    ENDPROC
    PROC Reflejado()
        MoveL Target_x_2,v100,z1,Marcador\WObj:=Pastel_2;
        MoveL Aproximacion_2,v100,z1,Marcador\WObj:=Pastel_2;
        MoveL HOME_2,v100,z1,Marcador\WObj:=Pastel_2;
        MoveL orientacioin_posible_2,v100,z1,Marcador\WObj:=Pastel_2;
        MoveL Target_10_2,v100,z1,Marcador\WObj:=Pastel_2;
        MoveL Target_20_2,v100,z1,Marcador\WObj:=Pastel_2;
        MoveL Target_30_2,v100,z1,Marcador\WObj:=Pastel_2;
        MoveL Target_40_2,v100,z1,Marcador\WObj:=Pastel_2;
        MoveL Target_50_2,v100,z1,Marcador\WObj:=Pastel_2;
        MoveL Target_60_2,v100,z1,Marcador\WObj:=Pastel_2;
        MoveL Target_70_2,v100,z1,Marcador\WObj:=Pastel_2;
        MoveL Target_80_2,v100,z1,Marcador\WObj:=Pastel_2;
        MoveL Target_90_2,v100,z1,Marcador\WObj:=Pastel_2;
        MoveL Target_100_2,v100,z1,Marcador\WObj:=Pastel_2;
        MoveL Target_110_2,v100,z1,Marcador\WObj:=Pastel_2;
        MoveL Target_120_2,v100,z1,Marcador\WObj:=Pastel_2;
        MoveL Target_130_2,v100,z1,Marcador\WObj:=Pastel_2;
        MoveL Target_140_2,v100,z1,Marcador\WObj:=Pastel_2;
        MoveL Target_150_2,v100,z1,Marcador\WObj:=Pastel_2;
        MoveL Target_160_2,v100,z1,Marcador\WObj:=Pastel_2;
        MoveL Target_170_2,v100,z1,Marcador\WObj:=Pastel_2;
        MoveL Target_180_2,v100,z1,Marcador\WObj:=Pastel_2;
        MoveL Target_190_2,v100,z1,Marcador\WObj:=Pastel_2;
        MoveL Target_200_2,v100,z1,Marcador\WObj:=Pastel_2;
        MoveL Target_210_2,v100,z1,Marcador\WObj:=Pastel_2;
        MoveL Target_220_2,v100,z1,Marcador\WObj:=Pastel_2;
        MoveL Target_230_2,v100,z1,Marcador\WObj:=Pastel_2;
        MoveL Target_240_2,v100,z1,Marcador\WObj:=Pastel_2;
        MoveL Target_250_2,v100,z1,Marcador\WObj:=Pastel_2;
        MoveL Target_260_2,v100,z1,Marcador\WObj:=Pastel_2;
        MoveL Target_270_2,v100,z1,Marcador\WObj:=Pastel_2;
        MoveL Target_280_2,v100,z1,Marcador\WObj:=Pastel_2;
        MoveL Target_290_2,v100,z1,Marcador\WObj:=Pastel_2;
        MoveL Target_300_2,v100,z1,Marcador\WObj:=Pastel_2;
        MoveL Target_310_2,v100,z1,Marcador\WObj:=Pastel_2;
        MoveL Target_320_2,v100,z1,Marcador\WObj:=Pastel_2;
        MoveL Target_330_2,v100,z1,Marcador\WObj:=Pastel_2;
        MoveL Target_340_2,v100,z1,Marcador\WObj:=Pastel_2;
        MoveL Target_350_2,v100,z1,Marcador\WObj:=Pastel_2;
        MoveL Target_360_2,v100,z1,Marcador\WObj:=Pastel_2;
        MoveL Target_370_2,v100,z1,Marcador\WObj:=Pastel_2;
        MoveL Target_380_2,v100,z1,Marcador\WObj:=Pastel_2;
        MoveL Target_390_2,v100,z1,Marcador\WObj:=Pastel_2;
        MoveL Target_400_2,v100,z1,Marcador\WObj:=Pastel_2;
        MoveL Target_410_2,v100,z1,Marcador\WObj:=Pastel_2;
        MoveL Target_420_2,v100,z1,Marcador\WObj:=Pastel_2;
        MoveL Target_430_2,v100,z1,Marcador\WObj:=Pastel_2;
        MoveL Target_440_2,v100,z1,Marcador\WObj:=Pastel_2;
        MoveL Target_450_2,v100,z1,Marcador\WObj:=Pastel_2;
        MoveL Target_460_2,v100,z1,Marcador\WObj:=Pastel_2;
        MoveL Target_470_2,v100,z1,Marcador\WObj:=Pastel_2;
        MoveL Target_480_2,v100,z1,Marcador\WObj:=Pastel_2;
        MoveL Target_490_2,v100,z1,Marcador\WObj:=Pastel_2;
        MoveL Target_500_2,v100,z1,Marcador\WObj:=Pastel_2;
        MoveL Target_510_2,v100,z1,Marcador\WObj:=Pastel_2;
        MoveL Target_520_2,v100,z1,Marcador\WObj:=Pastel_2;
        MoveL Target_530_2,v100,z1,Marcador\WObj:=Pastel_2;
        MoveL Target_540_2,v100,z1,Marcador\WObj:=Pastel_2;
        MoveL Target_550_2,v100,z1,Marcador\WObj:=Pastel_2;
        MoveL Target_560_2,v100,z1,Marcador\WObj:=Pastel_2;
        MoveL Target_570_2,v100,z1,Marcador\WObj:=Pastel_2;
        MoveL Target_580_2,v100,z1,Marcador\WObj:=Pastel_2;
        MoveL Target_590_2,v100,z1,Marcador\WObj:=Pastel_2;
        MoveL Target_600_2,v100,z1,Marcador\WObj:=Pastel_2;
        MoveL Target_610_2,v100,z1,Marcador\WObj:=Pastel_2;
        MoveL Target_620_2,v100,z1,Marcador\WObj:=Pastel_2;
        MoveL Target_630_2,v100,z1,Marcador\WObj:=Pastel_2;
        MoveL Target_640_2,v100,z1,Marcador\WObj:=Pastel_2;
        MoveL Target_650_2,v100,z1,Marcador\WObj:=Pastel_2;
        MoveL Target_660_2,v100,z1,Marcador\WObj:=Pastel_2;
        MoveL Target_670_2,v100,z1,Marcador\WObj:=Pastel_2;
        MoveL Target_680_2,v100,z1,Marcador\WObj:=Pastel_2;
        MoveL Target_690_2,v100,z1,Marcador\WObj:=Pastel_2;
        MoveL Target_700_2,v100,z1,Marcador\WObj:=Pastel_2;
        MoveL Target_710_2,v100,z1,Marcador\WObj:=Pastel_2;
        MoveL Target_720_2,v100,z1,Marcador\WObj:=Pastel_2;
        MoveL Target_730_2,v100,z1,Marcador\WObj:=Pastel_2;
        MoveL Target_740_2,v100,z1,Marcador\WObj:=Pastel_2;
        MoveL Target_750_2,v100,z1,Marcador\WObj:=Pastel_2;
        MoveL Target_760_2,v100,z1,Marcador\WObj:=Pastel_2;
        MoveL Target_770_2,v100,z1,Marcador\WObj:=Pastel_2;
        MoveL Target_780_2,v100,z1,Marcador\WObj:=Pastel_2;
        MoveL Target_790_2,v100,z1,Marcador\WObj:=Pastel_2;
        MoveL Target_800_2,v100,z1,Marcador\WObj:=Pastel_2;
        MoveL Target_810_2,v100,z1,Marcador\WObj:=Pastel_2;
        MoveL Target_820_2,v100,z1,Marcador\WObj:=Pastel_2;
        MoveL Target_830_2,v100,z1,Marcador\WObj:=Pastel_2;
        MoveL Target_840_2,v100,z1,Marcador\WObj:=Pastel_2;
        MoveL Target_850_2,v100,z1,Marcador\WObj:=Pastel_2;
        MoveL Target_860_2,v100,z1,Marcador\WObj:=Pastel_2;
        MoveL Target_870_2,v100,z1,Marcador\WObj:=Pastel_2;
        MoveL Target_880_2,v100,z1,Marcador\WObj:=Pastel_2;
        MoveL Target_890_2,v100,z1,Marcador\WObj:=Pastel_2;
        MoveL Target_900_2,v100,z1,Marcador\WObj:=Pastel_2;
        MoveL Target_910_2,v100,z1,Marcador\WObj:=Pastel_2;
        MoveL Target_920_2,v100,z1,Marcador\WObj:=Pastel_2;
        MoveL Target_930_2,v100,z1,Marcador\WObj:=Pastel_2;
        MoveL Target_940_2,v100,z1,Marcador\WObj:=Pastel_2;
        MoveL Target_950_2,v100,z1,Marcador\WObj:=Pastel_2;
        MoveL Target_960_2,v100,z1,Marcador\WObj:=Pastel_2;
        MoveL Target_970_2,v100,z1,Marcador\WObj:=Pastel_2;
        MoveL Target_980_2,v100,z1,Marcador\WObj:=Pastel_2;
        MoveL Target_990_2,v100,z1,Marcador\WObj:=Pastel_2;
        MoveL Target_1000_2,v100,z1,Marcador\WObj:=Pastel_2;
        MoveL Target_1010_2,v100,z1,Marcador\WObj:=Pastel_2;
        MoveL Target_1020_2,v100,z1,Marcador\WObj:=Pastel_2;
        MoveL Target_1030_2,v100,z1,Marcador\WObj:=Pastel_2;
        MoveL Target_1040_2,v100,z1,Marcador\WObj:=Pastel_2;
        MoveL Target_1050_2,v100,z1,Marcador\WObj:=Pastel_2;
        MoveL Target_1060_2,v100,z1,Marcador\WObj:=Pastel_2;
        MoveL Target_1070_2,v100,z1,Marcador\WObj:=Pastel_2;
        MoveL Target_1080_2,v100,z1,Marcador\WObj:=Pastel_2;
        MoveL Target_1090_2,v100,z1,Marcador\WObj:=Pastel_2;
        MoveL Target_1100_2,v100,z1,Marcador\WObj:=Pastel_2;
        MoveL Target_1110_2,v100,z1,Marcador\WObj:=Pastel_2;
        MoveL Target_1120_2,v100,z1,Marcador\WObj:=Pastel_2;
        MoveL Target_1130_2,v100,z1,Marcador\WObj:=Pastel_2;
        MoveL Target_1140_2,v100,z1,Marcador\WObj:=Pastel_2;
        MoveL Target_1150_2,v100,z1,Marcador\WObj:=Pastel_2;
        MoveL Target_1160_2,v100,z1,Marcador\WObj:=Pastel_2;
        MoveL Target_1170_2,v100,z1,Marcador\WObj:=Pastel_2;
        MoveL Target_1180_2,v100,z1,Marcador\WObj:=Pastel_2;
        MoveL Target_1190_2,v100,z1,Marcador\WObj:=Pastel_2;
        MoveL Target_1200_2,v100,z1,Marcador\WObj:=Pastel_2;
        MoveL Target_1210_2,v100,z1,Marcador\WObj:=Pastel_2;
        MoveL Target_1220_2,v100,z1,Marcador\WObj:=Pastel_2;
        MoveL Target_1230_2,v100,z1,Marcador\WObj:=Pastel_2;
        MoveL Target_1240_2,v100,z1,Marcador\WObj:=Pastel_2;
        MoveL Target_1250_2,v100,z1,Marcador\WObj:=Pastel_2;
        MoveL Target_1260_2,v100,z1,Marcador\WObj:=Pastel_2;
        MoveL Target_1270_2,v100,z1,Marcador\WObj:=Pastel_2;
        MoveL Target_1280_2,v100,z1,Marcador\WObj:=Pastel_2;
        MoveL Target_1290_2,v100,z1,Marcador\WObj:=Pastel_2;
        MoveL Target_1300_2,v100,z1,Marcador\WObj:=Pastel_2;
        MoveL Target_1310_2,v100,z1,Marcador\WObj:=Pastel_2;
        MoveL Target_1320_2,v100,z1,Marcador\WObj:=Pastel_2;
        MoveL Target_1330_2,v100,z1,Marcador\WObj:=Pastel_2;
        MoveL Target_1340_2,v100,z1,Marcador\WObj:=Pastel_2;
        MoveL Target_1350_2,v100,z1,Marcador\WObj:=Pastel_2;
        MoveL Target_1360_2,v100,z1,Marcador\WObj:=Pastel_2;
        MoveL Target_1370_2,v100,z1,Marcador\WObj:=Pastel_2;
        MoveL Target_1380_2,v100,z1,Marcador\WObj:=Pastel_2;
        MoveL Target_1390_2,v100,z1,Marcador\WObj:=Pastel_2;
        MoveL Target_1400_2,v100,z1,Marcador\WObj:=Pastel_2;
        MoveL Target_1410_2,v100,z1,Marcador\WObj:=Pastel_2;
        MoveL Target_1420_2,v100,z1,Marcador\WObj:=Pastel_2;
        MoveL Target_1430_2,v100,z1,Marcador\WObj:=Pastel_2;
        MoveL Target_1440_2,v100,z1,Marcador\WObj:=Pastel_2;
        MoveL Target_1450_2,v100,z1,Marcador\WObj:=Pastel_2;
        MoveL Target_1460_2,v100,z1,Marcador\WObj:=Pastel_2;
        MoveL Target_1470_2,v100,z1,Marcador\WObj:=Pastel_2;
        MoveL Target_1480_2,v100,z1,Marcador\WObj:=Pastel_2;
        MoveL Target_1490_2,v100,z1,Marcador\WObj:=Pastel_2;
        MoveL Target_1500_2,v100,z1,Marcador\WObj:=Pastel_2;
        MoveL Target_1510_2,v100,z1,Marcador\WObj:=Pastel_2;
        MoveL Target_1520_2,v100,z1,Marcador\WObj:=Pastel_2;
        MoveL Target_1530_2,v100,z1,Marcador\WObj:=Pastel_2;
        MoveL Target_1540_2,v100,z1,Marcador\WObj:=Pastel_2;
        MoveL Target_1550_2,v100,z1,Marcador\WObj:=Pastel_2;
        MoveL Target_1560_2,v100,z1,Marcador\WObj:=Pastel_2;
        MoveL Target_1570_2,v100,z1,Marcador\WObj:=Pastel_2;
        MoveL Target_1580_2,v100,z1,Marcador\WObj:=Pastel_2;
        MoveL Target_1590_2,v100,z1,Marcador\WObj:=Pastel_2;
        MoveL Target_1600_2,v100,z1,Marcador\WObj:=Pastel_2;
        MoveL Target_1610_2,v100,z1,Marcador\WObj:=Pastel_2;
        MoveL Target_1620_2,v100,z1,Marcador\WObj:=Pastel_2;
        MoveL Target_1630_2,v100,z1,Marcador\WObj:=Pastel_2;
        MoveL Target_1640_2,v100,z1,Marcador\WObj:=Pastel_2;
        MoveL Target_1650_2,v100,z1,Marcador\WObj:=Pastel_2;
        MoveL Target_1660_2,v100,z1,Marcador\WObj:=Pastel_2;
        MoveL Target_1670_2,v100,z1,Marcador\WObj:=Pastel_2;
        MoveL Target_1680_2,v100,z1,Marcador\WObj:=Pastel_2;
        MoveL Target_1690_2,v100,z1,Marcador\WObj:=Pastel_2;
        MoveL Target_1700_2,v100,z1,Marcador\WObj:=Pastel_2;
        MoveL Target_1710_2,v100,z1,Marcador\WObj:=Pastel_2;
        MoveL Target_1720_2,v100,z1,Marcador\WObj:=Pastel_2;
        MoveL Target_1730_2,v100,z1,Marcador\WObj:=Pastel_2;
        MoveL Target_1740_2,v100,z1,Marcador\WObj:=Pastel_2;
        MoveL Target_1750_2,v100,z1,Marcador\WObj:=Pastel_2;
        MoveL Target_1760_2,v100,z1,Marcador\WObj:=Pastel_2;
        MoveL Target_1770_2,v100,z1,Marcador\WObj:=Pastel_2;
        MoveL Target_1780_2,v100,z1,Marcador\WObj:=Pastel_2;
        MoveL Target_1790_2,v100,z1,Marcador\WObj:=Pastel_2;
        MoveL Target_1800_2,v100,z1,Marcador\WObj:=Pastel_2;
        MoveL Target_1810_2,v100,z1,Marcador\WObj:=Pastel_2;
        MoveL Target_1820_2,v100,z1,Marcador\WObj:=Pastel_2;
        MoveL Target_1830_2,v100,z1,Marcador\WObj:=Pastel_2;
        MoveL Target_1840_2,v100,z1,Marcador\WObj:=Pastel_2;
        MoveL Target_1850_2,v100,z1,Marcador\WObj:=Pastel_2;
        MoveL Target_1860_2,v100,z1,Marcador\WObj:=Pastel_2;
        MoveL Target_1870_2,v100,z1,Marcador\WObj:=Pastel_2;
        MoveL Target_1880_2,v100,z1,Marcador\WObj:=Pastel_2;
        MoveL Target_1890_2,v100,z1,Marcador\WObj:=Pastel_2;
        MoveL Target_1900_2,v100,z1,Marcador\WObj:=Pastel_2;
        MoveL Target_1910_2,v100,z1,Marcador\WObj:=Pastel_2;
        MoveL Target_1920_2,v100,z1,Marcador\WObj:=Pastel_2;
        MoveL Target_1930_2,v100,z1,Marcador\WObj:=Pastel_2;
        MoveL Target_1940_2,v100,z1,Marcador\WObj:=Pastel_2;
        MoveL Target_1950_2,v100,z1,Marcador\WObj:=Pastel_2;
        MoveL Target_1960_2,v100,z1,Marcador\WObj:=Pastel_2;
        MoveL Target_1970_2,v100,z1,Marcador\WObj:=Pastel_2;
        MoveL Target_1980_2,v100,z1,Marcador\WObj:=Pastel_2;
        MoveL Target_1990_2,v100,z1,Marcador\WObj:=Pastel_2;
        MoveL Target_2000_2,v100,z1,Marcador\WObj:=Pastel_2;
        MoveL Target_2010_2,v100,z1,Marcador\WObj:=Pastel_2;
        MoveL Target_2020_2,v100,z1,Marcador\WObj:=Pastel_2;
        MoveL Target_2030_2,v100,z1,Marcador\WObj:=Pastel_2;
        MoveL Target_2040_2,v100,z1,Marcador\WObj:=Pastel_2;
        MoveL Target_2050_2,v100,z1,Marcador\WObj:=Pastel_2;
        MoveL Target_2060_2,v100,z1,Marcador\WObj:=Pastel_2;
        MoveL Target_2070_2,v100,z1,Marcador\WObj:=Pastel_2;
        MoveL Target_2080_2,v100,z1,Marcador\WObj:=Pastel_2;
        MoveL Target_2090_2,v100,z1,Marcador\WObj:=Pastel_2;
        MoveL Target_2100_2,v100,z1,Marcador\WObj:=Pastel_2;
        MoveL Target_2110_2,v100,z1,Marcador\WObj:=Pastel_2;
        MoveL Target_2120_2,v100,z1,Marcador\WObj:=Pastel_2;
        MoveL Target_2130_2,v100,z1,Marcador\WObj:=Pastel_2;
        MoveL Target_2140_2,v100,z1,Marcador\WObj:=Pastel_2;
        MoveL Target_2150_2,v100,z1,Marcador\WObj:=Pastel_2;
        MoveL Target_2160_2,v100,z1,Marcador\WObj:=Pastel_2;
        MoveL Target_2170_2,v100,z1,Marcador\WObj:=Pastel_2;
        MoveL Target_2180_2,v100,z1,Marcador\WObj:=Pastel_2;
        MoveL Target_2190_2,v100,z1,Marcador\WObj:=Pastel_2;
        MoveL Target_2200_2,v100,z1,Marcador\WObj:=Pastel_2;
        MoveL Target_2210_2,v100,z1,Marcador\WObj:=Pastel_2;
        MoveL Target_2220_2,v100,z1,Marcador\WObj:=Pastel_2;
        MoveL Target_2230_2,v100,z1,Marcador\WObj:=Pastel_2;
        MoveL Target_2240_2,v100,z1,Marcador\WObj:=Pastel_2;
        MoveL Target_2250_2,v100,z1,Marcador\WObj:=Pastel_2;
        MoveL Target_2260_2,v100,z1,Marcador\WObj:=Pastel_2;
        MoveL Target_2270_2,v100,z1,Marcador\WObj:=Pastel_2;
        MoveL Target_2280_2,v100,z1,Marcador\WObj:=Pastel_2;
        MoveL Target_2290_2,v100,z1,Marcador\WObj:=Pastel_2;
        MoveL Target_2300_2,v100,z1,Marcador\WObj:=Pastel_2;
        MoveL Target_2310_2,v100,z1,Marcador\WObj:=Pastel_2;
        MoveL Target_2320_2,v100,z1,Marcador\WObj:=Pastel_2;
        MoveL Target_2330_2,v100,z1,Marcador\WObj:=Pastel_2;
        MoveL Target_2340_2,v100,z1,Marcador\WObj:=Pastel_2;
        MoveL Target_2350_2,v100,z1,Marcador\WObj:=Pastel_2;
        MoveL Target_2360_2,v100,z1,Marcador\WObj:=Pastel_2;
        MoveL Target_2370_2,v100,z1,Marcador\WObj:=Pastel_2;
        MoveL Target_2380_2,v100,z1,Marcador\WObj:=Pastel_2;
        MoveL Target_2390_2,v100,z1,Marcador\WObj:=Pastel_2;
        MoveL Target_2400_2,v100,z1,Marcador\WObj:=Pastel_2;
        MoveL Target_2410_2,v100,z1,Marcador\WObj:=Pastel_2;
        MoveL Target_2420_2,v100,z1,Marcador\WObj:=Pastel_2;
        MoveL Target_2430_2,v100,z1,Marcador\WObj:=Pastel_2;
        MoveL Target_2440_2,v100,z1,Marcador\WObj:=Pastel_2;
        MoveL Target_2450_2,v100,z1,Marcador\WObj:=Pastel_2;
        MoveL Target_2460_2,v100,z1,Marcador\WObj:=Pastel_2;
        MoveL Target_2470_2,v100,z1,Marcador\WObj:=Pastel_2;
        MoveL Target_2480_2,v100,z1,Marcador\WObj:=Pastel_2;
        MoveL Target_2490_2,v100,z1,Marcador\WObj:=Pastel_2;
        MoveL Target_2500_2,v100,z1,Marcador\WObj:=Pastel_2;
        MoveL Target_2510_2,v100,z1,Marcador\WObj:=Pastel_2;
        MoveL Target_2520_2,v100,z1,Marcador\WObj:=Pastel_2;
        MoveL Target_2530_2,v100,z1,Marcador\WObj:=Pastel_2;
        MoveL Target_2540_2,v100,z1,Marcador\WObj:=Pastel_2;
        MoveL Target_2550_2,v100,z1,Marcador\WObj:=Pastel_2;
        MoveL Target_2560_2,v100,z1,Marcador\WObj:=Pastel_2;
        MoveL Target_2570_2,v100,z1,Marcador\WObj:=Pastel_2;
        MoveL Target_2580_2,v100,z1,Marcador\WObj:=Pastel_2;
        MoveL Target_2590_2,v100,z1,Marcador\WObj:=Pastel_2;
        MoveL Target_2600_2,v100,z1,Marcador\WObj:=Pastel_2;
        MoveL Target_2610_2,v100,z1,Marcador\WObj:=Pastel_2;
        MoveL Target_2620_2,v100,z1,Marcador\WObj:=Pastel_2;
        MoveL Target_2630_2,v100,z1,Marcador\WObj:=Pastel_2;
        MoveL Target_2640_2,v100,z1,Marcador\WObj:=Pastel_2;
        MoveL Target_2650_2,v100,z1,Marcador\WObj:=Pastel_2;
        MoveL Target_2660_2,v100,z1,Marcador\WObj:=Pastel_2;
        MoveL Target_2670_2,v100,z1,Marcador\WObj:=Pastel_2;
        MoveL Target_2680_2,v100,z1,Marcador\WObj:=Pastel_2;
        MoveL Target_2690_2,v100,z1,Marcador\WObj:=Pastel_2;
        MoveL Target_2700_2,v100,z1,Marcador\WObj:=Pastel_2;
        MoveL Target_2710_2,v100,z1,Marcador\WObj:=Pastel_2;
        MoveL Target_2720_2,v100,z1,Marcador\WObj:=Pastel_2;
        MoveL Target_2730_2,v100,z1,Marcador\WObj:=Pastel_2;
        MoveL Target_2740_2,v100,z1,Marcador\WObj:=Pastel_2;
        MoveL Target_2750_2,v100,z1,Marcador\WObj:=Pastel_2;
        MoveL Target_2760_2,v100,z1,Marcador\WObj:=Pastel_2;
        MoveL Target_2770_2,v100,z1,Marcador\WObj:=Pastel_2;
        MoveL Target_2780_2,v100,z1,Marcador\WObj:=Pastel_2;
        MoveL Target_2790_2,v100,z1,Marcador\WObj:=Pastel_2;
        MoveL Target_2800_2,v100,z1,Marcador\WObj:=Pastel_2;
        MoveL Target_2810_2,v100,z1,Marcador\WObj:=Pastel_2;
        MoveL Target_2820_2,v100,z1,Marcador\WObj:=Pastel_2;
        MoveL Target_2830_2,v100,z1,Marcador\WObj:=Pastel_2;
        MoveL Target_2840_2,v100,z1,Marcador\WObj:=Pastel_2;
        MoveL Target_2850_2,v100,z1,Marcador\WObj:=Pastel_2;
        MoveL Target_2860_2,v100,z1,Marcador\WObj:=Pastel_2;
        MoveL Target_2870_2,v100,z1,Marcador\WObj:=Pastel_2;
        MoveL Target_2880_2,v100,z1,Marcador\WObj:=Pastel_2;
        MoveL Target_2890_2,v100,z1,Marcador\WObj:=Pastel_2;
        MoveL Target_2900_2,v100,z1,Marcador\WObj:=Pastel_2;
        MoveL Target_2910_2,v100,z1,Marcador\WObj:=Pastel_2;
        MoveL Target_2920_2,v100,z1,Marcador\WObj:=Pastel_2;
        MoveL Target_2930_2,v100,z1,Marcador\WObj:=Pastel_2;
        MoveL Target_2940_2,v100,z1,Marcador\WObj:=Pastel_2;
        MoveL Target_2950_2,v100,z1,Marcador\WObj:=Pastel_2;
        MoveL Target_2960_2,v100,z1,Marcador\WObj:=Pastel_2;
        MoveL Target_2970_2,v100,z1,Marcador\WObj:=Pastel_2;
        MoveL Target_2980_2,v100,z1,Marcador\WObj:=Pastel_2;
        MoveL Target_2990_2,v100,z1,Marcador\WObj:=Pastel_2;
        MoveL Target_3000_2,v100,z1,Marcador\WObj:=Pastel_2;
        MoveL Target_3010_2,v100,z1,Marcador\WObj:=Pastel_2;
        MoveL Target_3020_2,v100,z1,Marcador\WObj:=Pastel_2;
        MoveL Target_3030_2,v100,z1,Marcador\WObj:=Pastel_2;
        MoveL Target_3040_2,v100,z1,Marcador\WObj:=Pastel_2;
        MoveL Target_3050_2,v100,z1,Marcador\WObj:=Pastel_2;
        MoveL Target_3060_2,v100,z1,Marcador\WObj:=Pastel_2;
        MoveL Target_3070_2,v100,z1,Marcador\WObj:=Pastel_2;
        MoveL Target_3080_2,v100,z1,Marcador\WObj:=Pastel_2;
        MoveL Target_3090_2,v100,z1,Marcador\WObj:=Pastel_2;
        MoveL Target_3100_2,v100,z1,Marcador\WObj:=Pastel_2;
        MoveL Target_3110_2,v100,z1,Marcador\WObj:=Pastel_2;
        MoveL Target_3120_2,v100,z1,Marcador\WObj:=Pastel_2;
        MoveL Target_3130_2,v100,z1,Marcador\WObj:=Pastel_2;
        MoveL Target_3140_2,v100,z1,Marcador\WObj:=Pastel_2;
        MoveL Target_3150_2,v100,z1,Marcador\WObj:=Pastel_2;
        MoveL Target_3160_2,v100,z1,Marcador\WObj:=Pastel_2;
        MoveL Target_3170_2,v100,z1,Marcador\WObj:=Pastel_2;
        MoveL Target_3180_2,v100,z1,Marcador\WObj:=Pastel_2;
        MoveL Target_3190_2,v100,z1,Marcador\WObj:=Pastel_2;
        MoveL Target_3200_2,v100,z1,Marcador\WObj:=Pastel_2;
        MoveL Target_3210_2,v100,z1,Marcador\WObj:=Pastel_2;
        MoveL Target_3220_2,v100,z1,Marcador\WObj:=Pastel_2;
        MoveL Target_3230_2,v100,z1,Marcador\WObj:=Pastel_2;
        MoveL Target_3240_2,v100,z1,Marcador\WObj:=Pastel_2;
        MoveL Target_3250_2,v100,z1,Marcador\WObj:=Pastel_2;
        MoveL Target_3260_2,v100,z1,Marcador\WObj:=Pastel_2;
        MoveL Target_3270_2,v100,z1,Marcador\WObj:=Pastel_2;
        MoveL Target_3280_2,v100,z1,Marcador\WObj:=Pastel_2;
        MoveL Target_3290_2,v100,z1,Marcador\WObj:=Pastel_2;
        MoveL Target_3300_2,v100,z1,Marcador\WObj:=Pastel_2;
        MoveL Target_3310_2,v100,z1,Marcador\WObj:=Pastel_2;
        MoveL Target_3320_2,v100,z1,Marcador\WObj:=Pastel_2;
        MoveL Target_3330_2,v100,z1,Marcador\WObj:=Pastel_2;
        MoveL Target_3340_2,v100,z1,Marcador\WObj:=Pastel_2;
        MoveL Target_3350_2,v100,z1,Marcador\WObj:=Pastel_2;
        MoveL Target_3360_2,v100,z1,Marcador\WObj:=Pastel_2;
        MoveL Target_3370_2,v100,z1,Marcador\WObj:=Pastel_2;
        MoveL Target_3380_2,v100,z1,Marcador\WObj:=Pastel_2;
        MoveL Target_3390_2,v100,z1,Marcador\WObj:=Pastel_2;
        MoveL Target_3400_2,v100,z1,Marcador\WObj:=Pastel_2;
        MoveL Target_3410_2,v100,z1,Marcador\WObj:=Pastel_2;
        MoveL Target_3420_2,v100,z1,Marcador\WObj:=Pastel_2;
        MoveL Target_3430_2,v100,z1,Marcador\WObj:=Pastel_2;
        MoveL Target_3440_2,v100,z1,Marcador\WObj:=Pastel_2;
        MoveL Target_3450_2,v100,z1,Marcador\WObj:=Pastel_2;
        MoveL Target_3460_2,v100,z1,Marcador\WObj:=Pastel_2;
        MoveL Target_3470_2,v100,z1,Marcador\WObj:=Pastel_2;
        MoveL Target_3480_2,v100,z1,Marcador\WObj:=Pastel_2;
        MoveL Target_3490_2,v100,z1,Marcador\WObj:=Pastel_2;
        MoveL Target_3500_2,v100,z1,Marcador\WObj:=Pastel_2;
        MoveL Target_3510_2,v100,z1,Marcador\WObj:=Pastel_2;
        MoveL Target_3520_2,v100,z1,Marcador\WObj:=Pastel_2;
        MoveL Target_3530_2,v100,z1,Marcador\WObj:=Pastel_2;
        MoveL Target_3540_2,v100,z1,Marcador\WObj:=Pastel_2;
        MoveL Target_3550_2,v100,z1,Marcador\WObj:=Pastel_2;
        MoveL Target_3560_2,v100,z1,Marcador\WObj:=Pastel_2;
        MoveL Target_3570_2,v100,z1,Marcador\WObj:=Pastel_2;
        MoveL Target_3580_2,v100,z1,Marcador\WObj:=Pastel_2;
        MoveL Target_3590_2,v100,z1,Marcador\WObj:=Pastel_2;
        MoveL Target_3600_2,v100,z1,Marcador\WObj:=Pastel_2;
        MoveL Target_3610_2,v100,z1,Marcador\WObj:=Pastel_2;
        MoveL Target_3620_2,v100,z1,Marcador\WObj:=Pastel_2;
        MoveL Target_3630_2,v100,z1,Marcador\WObj:=Pastel_2;
        MoveL Target_3640_2,v100,z1,Marcador\WObj:=Pastel_2;
        MoveL Target_3650_2,v100,z1,Marcador\WObj:=Pastel_2;
        MoveL Target_3660_2,v100,z1,Marcador\WObj:=Pastel_2;
        MoveL Target_3670_2,v100,z1,Marcador\WObj:=Pastel_2;
        MoveL Target_3680_2,v100,z1,Marcador\WObj:=Pastel_2;
        MoveL Target_3690_2,v100,z1,Marcador\WObj:=Pastel_2;
        MoveL Target_3700_2,v100,z1,Marcador\WObj:=Pastel_2;
        MoveL Target_3710_2,v100,z1,Marcador\WObj:=Pastel_2;
        MoveL Target_3720_2,v100,z1,Marcador\WObj:=Pastel_2;
        MoveL Target_3730_2,v100,z1,Marcador\WObj:=Pastel_2;
        MoveL Target_3740_2,v100,z1,Marcador\WObj:=Pastel_2;
        MoveL Target_3750_2,v100,z1,Marcador\WObj:=Pastel_2;
        MoveL Target_3760_2,v100,z1,Marcador\WObj:=Pastel_2;
        MoveL Target_3770_2,v100,z1,Marcador\WObj:=Pastel_2;
        MoveL Target_3780_2,v100,z1,Marcador\WObj:=Pastel_2;
        MoveL Target_3790_2,v100,z1,Marcador\WObj:=Pastel_2;
        MoveL Target_3800_2,v100,z1,Marcador\WObj:=Pastel_2;
        MoveL Target_3810_2,v100,z1,Marcador\WObj:=Pastel_2;
        MoveL Target_3820_2,v100,z1,Marcador\WObj:=Pastel_2;
        MoveL Target_3830_2,v100,z1,Marcador\WObj:=Pastel_2;
        MoveL Target_3840_2,v100,z1,Marcador\WObj:=Pastel_2;
        MoveL Target_3850_2,v100,z1,Marcador\WObj:=Pastel_2;
        MoveL Target_3860_2,v100,z1,Marcador\WObj:=Pastel_2;
        MoveL Target_3870_2,v100,z1,Marcador\WObj:=Pastel_2;
        MoveL Target_3880_2,v100,z1,Marcador\WObj:=Pastel_2;
        MoveL Target_3890_2,v100,z1,Marcador\WObj:=Pastel_2;
        MoveL Target_3900_2,v100,z1,Marcador\WObj:=Pastel_2;
        MoveL Target_3910_2,v100,z1,Marcador\WObj:=Pastel_2;
        MoveL Target_3920_2,v100,z1,Marcador\WObj:=Pastel_2;
        MoveL Target_3930_2,v100,z1,Marcador\WObj:=Pastel_2;
        MoveL Target_3940_2,v100,z1,Marcador\WObj:=Pastel_2;
    ENDPROC
ENDMODULE
